Staubli VAL3: AXISMOVEL.pjx

--- AXISMOVEL.pjx ---
Parameters version=s7.2.1 stackSize=5000 millimeterUnit=true
Program file=find.pgx
Program file=get.pgx
Program file=getSize.pgx
Program file=loadCycle.pgx
Program file=onEdit.pgx
Program file=onInsert.pgx
Program file=onProgEnd.pgx
Program file=onRun.pgx
Program file=onStart.pgx
Program file=onStop.pgx
Data file=AXISMOVEL.dtx
Library alias=io path=Disk://io/io.pjx
Library alias=use path=Disk://kernel/userPage/userPage.pjx

--- find.pgx ---
public program find(string& x_sItem[], bool& x_bFound[])
begin
end

--- getSize.pgx ---
public program getSize(num& x_nSize[])
begin
end

--- loadCycle.pgx ---
public program loadCycle(string& x_sName[], num& x_nResult[])
begin
  //
  // load the select program for the Cycle
  //
end

--- onEdit.pgx ---
public program onEdit(string& x_sItem[])
  local num l_nX
  local num l_nY
  local num l_nDelay
begin
  // convert to a num
  toNum(x_sItem,l_nDelay,true)
  // change the field
  call use:insertDialog("Distance [mm] ",l_nDelay,-0.01,2680.01)
  // give back
  if l_nDelay>=0
    l_nDelay=round(l_nDelay)
    x_sItem="AXISMOVEL "+toString("",l_nDelay)
  endIf
end

--- onInsert.pgx ---
public program onInsert(string& x_sItem[])
  local num l_nDelay
begin
  cls()
  l_nDelay=0
  call use:insertDialog("Distance [mm] ",l_nDelay,-0.01,2680.01)
  // give back
  if l_nDelay>=0
    l_nDelay=round(l_nDelay)
    x_sItem="AXISMOVEL "+toString("",l_nDelay)
  endIf
end

--- onProgEnd.pgx ---
public program onProgEnd(string& x_sItem[])
begin
end

--- onRun.pgx ---
public program onRun(string& x_sItem[])
  local num l_nValue
  local num l_nVelocity
begin
  //
  // convert to a num
  if aioGet(io:MbAI_bBackHome)!=1
    popUpMsg("7轴未回零位，请先执行回零操作！")
    return
  endIf
  if !isPowered()
    popUpMsg("请给手臂上电")
    return
  endIf
  bAxisMove=true
  aioSet(io:MbAO_b7Axis,1)
  aioSet(io:MbAO_bMoveToPos,0)
  toNum(x_sItem,l_nValue,true)
  // NB the robot will no STOP
//  aioSet(io:MbAI_bAxis7Reac,0)
  delay(0.5)
  l_nVelocity=speedScale()
  l_nVelocity=700*l_nVelocity/100
  l_nVelocity=round(l_nVelocity)
  l_nValue=round(l_nValue)
  aioSet(io:MbAO_aMovePosL,0)
  aioSet(io:MbAO_aMovePosH,2.554265*l_nValue)
  aioSet(io:MbAO_aMoveDis,1)
  aioSet(io:MbAO_aVelocity,l_nVelocity)
  aioSet(io:MbAO_bMoveToPos,1)
  delay(0.5)
  wait(aioGet(io:MbAI_bAxis7Reac)==0)
  wait(aioGet(io:MbAI_bAxis7Reac)==1)
  aioSet(io:MbAO_bMoveToPos,0)
  aioSet(io:MbAO_aMoveDis,0)
  aioSet(io:MbAO_b7Axis,0)
  logMsg("6")
  bAxisMove=false
end

--- onStop.pgx ---
public program onStop(string& x_sItem[])
begin
  aioSet(io:MbAO_aMoveDis,0)
  aioSet(io:MbAO_b7Axis,0)
  logMsg("7")
end
